Omron CX-Programmer project NewProject (CX-Programmer 9.75)

# PLC NewPLC1: CP2E-N N

## Program NewProgram1 (cyclic task 0)

### Section Section1

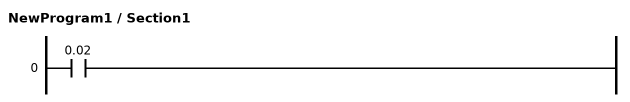
; rung 0
LD 0.02

### Section END
; rung 0
END(001)